// Mitsubishi GX Works2 project: 과정 평가 문항 1   PLC: Q03UDV

PROGRAM MAIN
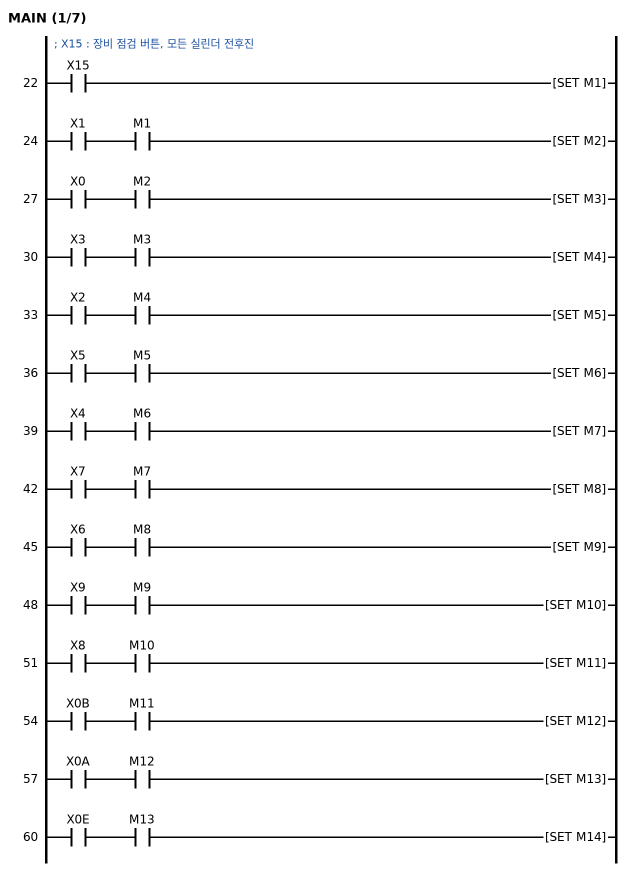
; X15 : 장비 점검 버튼, 모든 실린더 전후진
22    LD      X15
      SET     M1
24    LD      X1
      AND     M1
      SET     M2
27    LD      X0
      AND     M2
      SET     M3
30    LD      X3
      AND     M3
      SET     M4
33    LD      X2
      AND     M4
      SET     M5
36    LD      X5
      AND     M5
      SET     M6
39    LD      X4
      AND     M6
      SET     M7
42    LD      X7
      AND     M7
      SET     M8
45    LD      X6
      AND     M8
      SET     M9
48    LD      X9
      AND     M9
      SET     M10
51    LD      X8
      AND     M10
      SET     M11
54    LD      X0B
      AND     M11
      SET     M12
57    LD      X0A
      AND     M12
      SET     M13
60    LD      X0E
      AND     M13
      SET     M14
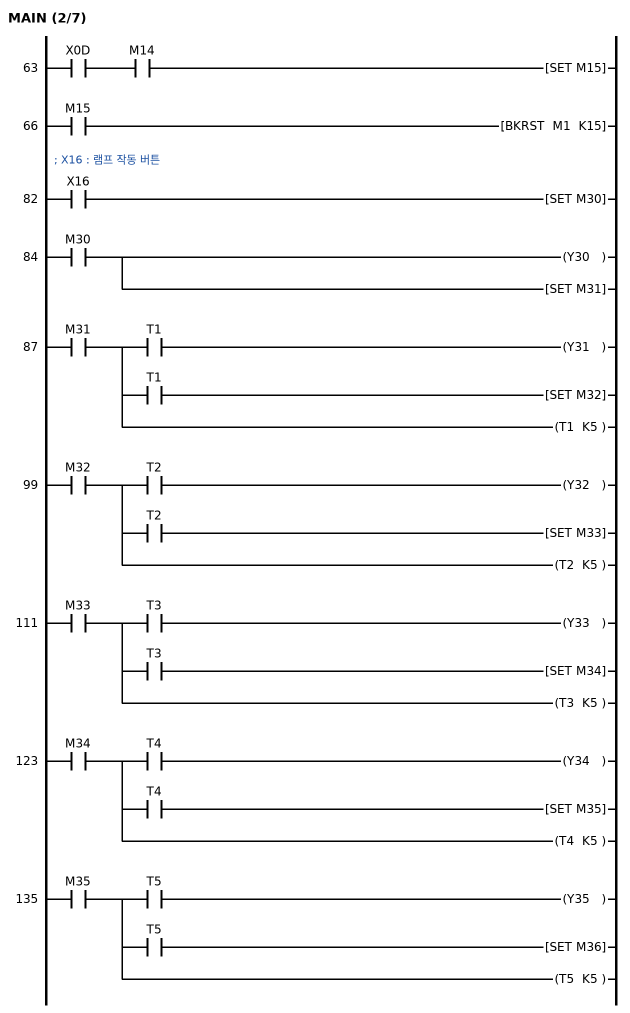
63    LD      X0D
      AND     M14
      SET     M15
66    LD      M15
      BKRST   M1 K15
; X16 : 램프 작동 버튼
82    LD      X16
      SET     M30
84    LD      M30
      OUT     Y30
      SET     M31
87    LD      M31
      MPS
      AND     T1
      OUT     Y31
      MRD
      AND     T1
      SET     M32
      MPP
      OUT     T1 K5
99    LD      M32
      MPS
      AND     T2
      OUT     Y32
      MRD
      AND     T2
      SET     M33
      MPP
      OUT     T2 K5
111   LD      M33
      MPS
      AND     T3
      OUT     Y33
      MRD
      AND     T3
      SET     M34
      MPP
      OUT     T3 K5
123   LD      M34
      MPS
      AND     T4
      OUT     Y34
      MRD
      AND     T4
      SET     M35
      MPP
      OUT     T4 K5
135   LD      M35
      MPS
      AND     T5
      OUT     Y35
      MRD
      AND     T5
      SET     M36
      MPP
      OUT     T5 K5
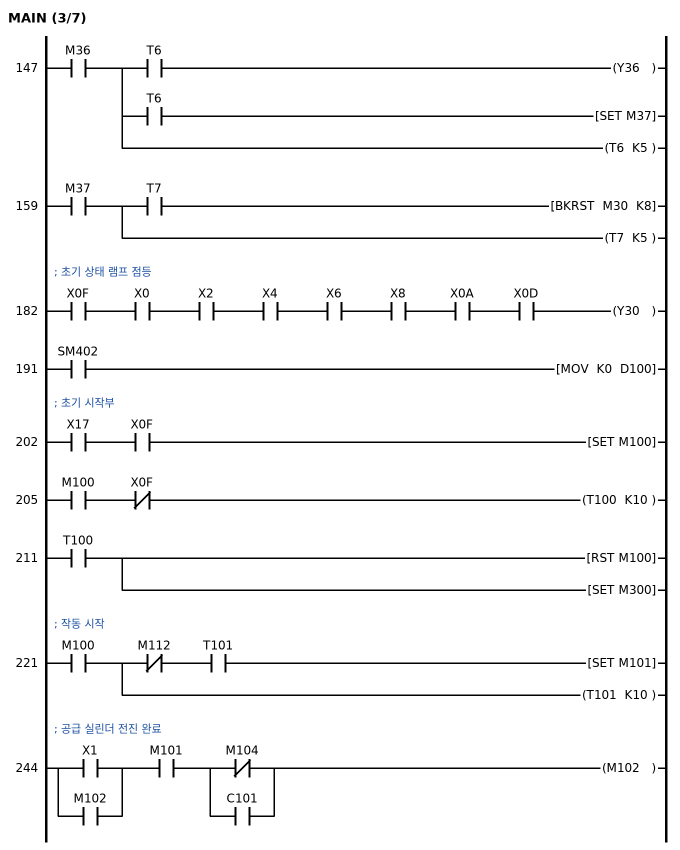
147   LD      M36
      MPS
      AND     T6
      OUT     Y36
      MRD
      AND     T6
      SET     M37
      MPP
      OUT     T6 K5
159   LD      M37
      MPS
      AND     T7
      BKRST   M30 K8
      MPP
      OUT     T7 K5
; 초기 상태 램프 점등
182   LD      X0F
      AND     X0
      AND     X2
      AND     X4
      AND     X6
      AND     X8
      AND     X0A
      AND     X0D
      OUT     Y30
191   LD      SM402
      MOV     K0 D100
; 초기 시작부
202   LD      X17
      AND     X0F
      SET     M100
205   LD      M100
      ANI     X0F
      OUT     T100 K10
211   LD      T100
      RST     M100
      SET     M300
; 작동 시작
221   LD      M100
      MPS
      ANI     M112
      AND     T101
      SET     M101
      MPP
      OUT     T101 K10
; 공급 실린더 전진 완료
244   LD      X1
      OR      M102
      AND     M101
      LDI     M104
      OR      C101
      ANB
      OUT     M102
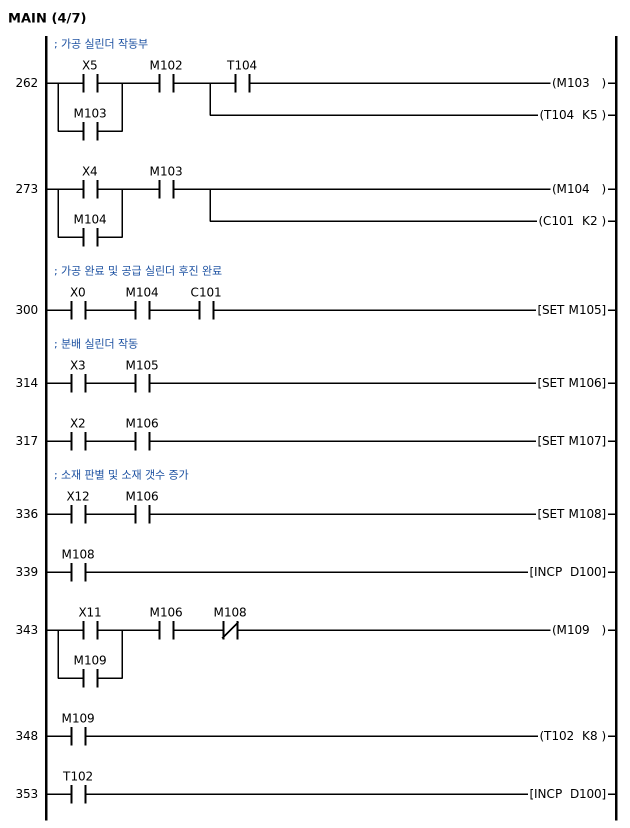
; 가공 실린더 작동부
262   LD      X5
      OR      M103
      AND     M102
      MPS
      AND     T104
      OUT     M103
      MPP
      OUT     T104 K5
273   LD      X4
      OR      M104
      AND     M103
      OUT     M104
      OUT     C101 K2
; 가공 완료 및 공급 실린더 후진 완료
300   LD      X0
      AND     M104
      AND     C101
      SET     M105
; 분배 실린더 작동
314   LD      X3
      AND     M105
      SET     M106
317   LD      X2
      AND     M106
      SET     M107
; 소재 판별 및 소재 갯수 증가
336   LD      X12
      AND     M106
      SET     M108
339   LD      M108
      INCP    D100
343   LD      X11
      OR      M109
      AND     M106
      ANI     M108
      OUT     M109
348   LD      M109
      OUT     T102 K8
353   LD      T102
      INCP    D100
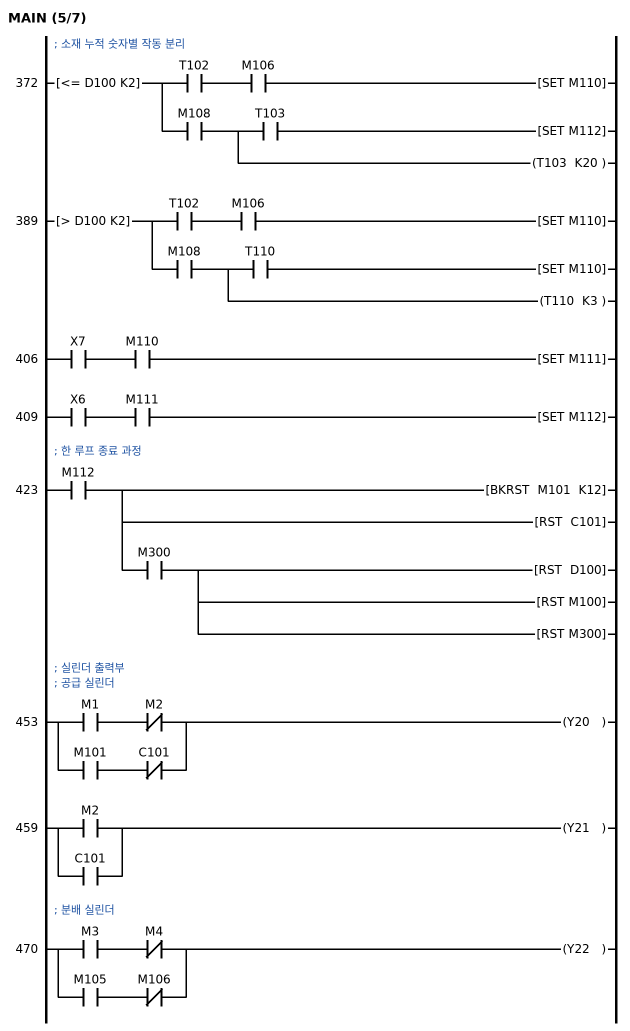
; 소재 누적 숫자별 작동 분리
372   LD<=    D100 K2
      MPS
      AND     T102
      AND     M106
      SET     M110
      MPP
      AND     M108
      MPS
      AND     T103
      SET     M112
      MPP
      OUT     T103 K20
389   LD>     D100 K2
      MPS
      AND     T102
      AND     M106
      SET     M110
      MPP
      AND     M108
      MPS
      AND     T110
      SET     M110
      MPP
      OUT     T110 K3
406   LD      X7
      AND     M110
      SET     M111
409   LD      X6
      AND     M111
      SET     M112
; 한 루프 종료 과정
423   LD      M112
      BKRST   M101 K12
      RST     C101
      AND     M300
      RST     D100
      RST     M100
      RST     M300
; 실린더 출력부
; 공급 실린더
453   LD      M1
      ANI     M2
      LD      M101
      ANI     C101
      ORB
      OUT     Y20
459   LD      M2
      OR      C101
      OUT     Y21
; 분배 실린더
470   LD      M3
      ANI     M4
      LD      M105
      ANI     M106
      ORB
      OUT     Y22
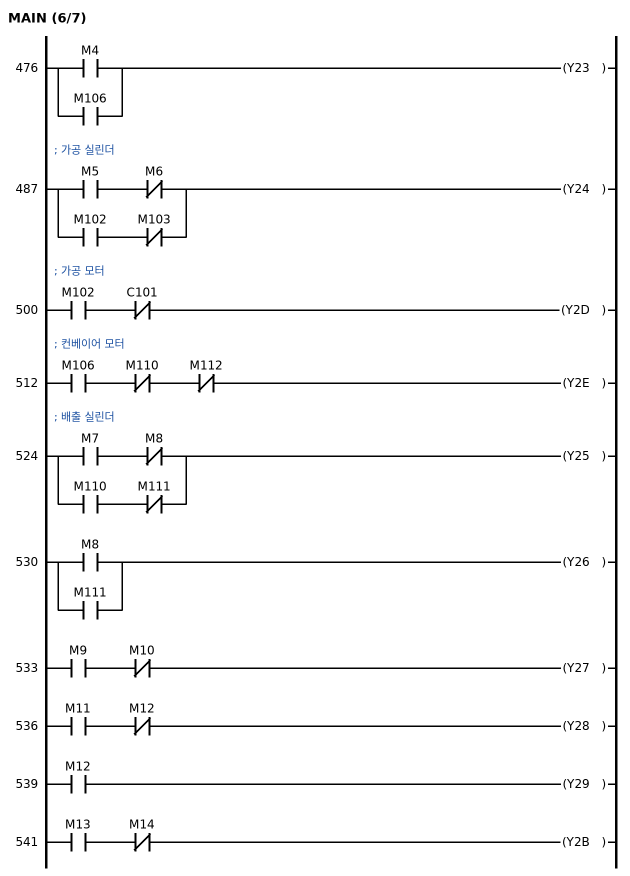
476   LD      M4
      OR      M106
      OUT     Y23
; 가공 실린더
487   LD      M5
      ANI     M6
      LD      M102
      ANI     M103
      ORB
      OUT     Y24
; 가공 모터
500   LD      M102
      ANI     C101
      OUT     Y2D
; 컨베이어 모터
512   LD      M106
      ANI     M110
      ANI     M112
      OUT     Y2E
; 배출 실린더
524   LD      M7
      ANI     M8
      LD      M110
      ANI     M111
      ORB
      OUT     Y25
530   LD      M8
      OR      M111
      OUT     Y26
533   LD      M9
      ANI     M10
      OUT     Y27
536   LD      M11
      ANI     M12
      OUT     Y28
539   LD      M12
      OUT     Y29
541   LD      M13
      ANI     M14
      OUT     Y2B
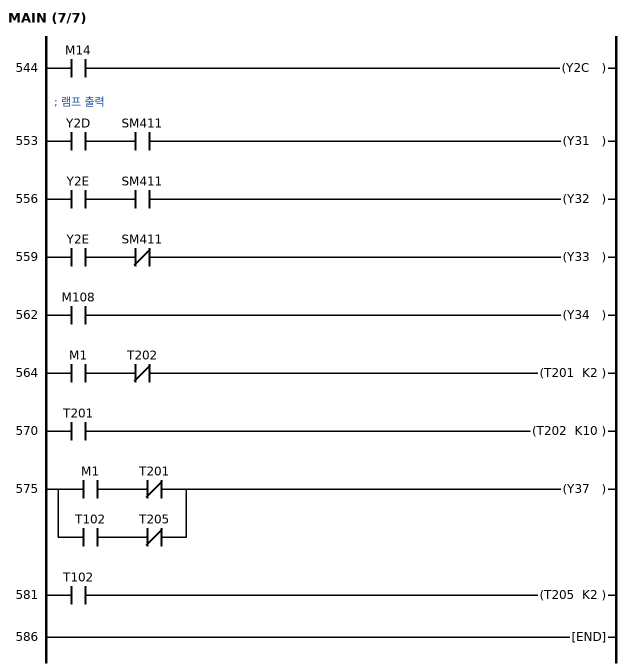
544   LD      M14
      OUT     Y2C
; 램프 출력
553   LD      Y2D
      AND     SM411
      OUT     Y31
556   LD      Y2E
      AND     SM411
      OUT     Y32
559   LD      Y2E
      ANI     SM411
      OUT     Y33
562   LD      M108
      OUT     Y34
564   LD      M1
      ANI     T202
      OUT     T201 K2
570   LD      T201
      OUT     T202 K10
575   LD      M1
      ANI     T201
      LD      T102
      ANI     T205
      ORB
      OUT     Y37
581   LD      T102
      OUT     T205 K2
586   END
END_PROGRAM
